// TwinCAT 3 PLC project IBF_System
// Title: IBF_System
// Company: Industrial Brains B.V.
// ProjectVersion: 0.0.0.0
// Description: system and module base functions
// ProgramVersion: 3.1.4023.0
// libraries:
//   IBF_Devices, * (Industrial Brains B.V.)
//   IBF_HMI, * (Industrial Brains B.V.)
//   IBF_Utilities, * (Industrial Brains B.V.)
//   Tc2_Standard, * (Beckhoff Automation GmbH)
//   Tc2_System, * (Beckhoff Automation GmbH)
//   Tc2_Utilities, * (Beckhoff Automation GmbH)
//   Tc3_Module, * (Beckhoff Automation GmbH)
// project tree:
//   GVLs/ PAR_System.TcGVL, GVL_System.TcGVL
//   / PlcTask.TcTTO
//   FaultHandler/ Fb_SystemFaultHandler.TcPOU (excluded from build)
//   ModuleBase/Base/ Fb_ModuleBase.TcPOU
//   SystemBase/DataTypes/ E_StateSystem.TcTLEO, Udt_ModuleId.TcDUT
//   SystemBase/ SystemBase.TcPOU
//   _TESTS/ FB_DummyModule.TcPOU, PRG_TEST.TcPOU

CONFIGURATION IBF_System
    RESOURCE PLC ON TwinCAT3
        TASK PlcTask(INTERVAL := T#10ms, PRIORITY := 6);
        PROGRAM PRG_TEST WITH PlcTask : PRG_TEST;
    END_RESOURCE
END_CONFIGURATION

// ---- SystemBase/DataTypes/E_StateSystem.TcTLEO
{attribute 'qualified_only'}
{attribute 'strict'}
{attribute 'to_string'}
TYPE E_StateSystem :
(
	FirstCycle		,
	CheckLogger		,
	CheckReferences ,  	// System is checking if module references are OK
	Initialize		, 	// System is initializing
	LoadParameters	, 	// System is loading parameters from/to file
	Safe			, 	// System is in safety state
	Enable			, 	// System is enabling 
	Home			, 	// system is homing 
	Resetting		, 	// System is resetting
	Idle			, 	// system is waiting for commands
	Manual			, 	// System is in manual mode
	SemiAuto		, 	// System is in semi auto mode
	Automatic		, 	// system is in automatic mode 
	Fault				// System is in Fault state
) UDINT;
END_TYPE

// ---- SystemBase/DataTypes/Udt_ModuleId.TcDUT
TYPE Udt_ModuleId :
STRUCT
	nNumber		: UDINT ; // Module identification number used for sorting order
	sName		: STRING; // Module name
	pFunction	: POINTER TO Fb_ModuleBase ;
END_STRUCT
END_TYPE

// ---- GVLs/PAR_System.TcGVL
{attribute 'qualified_only'}
VAR_GLOBAL CONSTANT
	LOG_FOLDER : STRING := ''; // Location for the log files
END_VAR

// ---- GVLs/GVL_System.TcGVL

{attribute 'qualified_only'} // Main system variables and state indicators
{attribute 'analysis':= '-33'}
VAR_GLOBAL CONSTANT
	cnMaxNUMBEROFMODULES 	: UDINT := 10 		; // "maximum" number of modules in the system
	CtAIRPRESSUREDELAY	: TIME 	:= T#500MS	; // Timout before air fault becomes active
	cbUPSPRESENT		: BOOL	:= FALSE 	; // Enable automatic shutdown when power is interupted
END_VAR
VAR_GLOBAL PERSISTENT
	nTotalUnitsProduced		: UDINT ; // Units produced 
END_VAR

// ---- _TESTS/PRG_TEST.TcPOU
PROGRAM INTERNAL PRG_TEST
VAR
 	bEnableTests : BOOL;

	fbDummyModule : FB_DummyModule;
END_VAR

IF bEnableTests THEN
	// SystemBase is the master program. it controls all underlying modules.
	SystemBase();

	// Call modules
	fbDummyModule(nModuleID:= 1);
END_IF

END_PROGRAM

// ---- _TESTS/FB_DummyModule.TcPOU
FUNCTION_BLOCK INTERNAL FB_DummyModule EXTENDS Fb_ModuleBase
VAR_INPUT
	// Inputs for testing module <> system interaction
	bAllowInit 		: BOOL;
	bAllowAutomatic : BOOL;
	bAllowSemiAuto 	: BOOL;
	bAllowHold 		: BOOL;
	bAllowHome 		: BOOL;
	bAllowReset 	: BOOL;
	bAllowIsSafe 	: BOOL;
	bAllowManual 	: BOOL;
END_VAR
VAR
	nCallsToExecAutomatic : ULINT;
	nCallsToExecHold : ULINT;
	nCallsToExecHome : ULINT;
	nCallsToExecInit : ULINT;
	nCallsToExecManual : ULINT;
	nCallsToExecReset : ULINT;
	nCallsToExecSafeStop : ULINT;
	nCallsToExecSemiAuto : ULINT;
END_VAR

SUPER^();

METHOD PROTECTED  CallComponents : BOOL
VAR_INPUT
END_VAR
END_METHOD

METHOD PROTECTED  CheckCollision : BOOL // Checks device commands for positble collisions  and block if necesarry
VAR_INPUT
END_VAR
END_METHOD

METHOD PROTECTED  ExecAutomatic : BOOL
VAR_INPUT
END_VAR
bAutomatic := bAllowAutomatic;
ExecAutomatic := bAutomatic;

nCallsToExecAutomatic := nCallsToExecAutomatic + 1;
END_METHOD

METHOD PROTECTED  ExecBaseFunctions : BOOL
VAR_INPUT
END_VAR
END_METHOD

METHOD PROTECTED  ExecEnable
VAR_INPUT
END_VAR
END_METHOD

METHOD PROTECTED  ExecHold : BOOL
VAR_INPUT
END_VAR
bHeld := bAllowHold;
ExecHold := bHeld;

nCallsToExecHold := nCallsToExecHold + 1;
END_METHOD

METHOD PROTECTED  ExecHome : BOOL
VAR_INPUT
END_VAR
bHomed := bAllowHome;
ExecHome := bHomed;

nCallsToExecHome := nCallsToExecHome + 1;
END_METHOD

METHOD PROTECTED  ExecIdle
VAR_INPUT
END_VAR
END_METHOD

METHOD PROTECTED  ExecInit : BOOL
VAR_INPUT
END_VAR
bInitialized := bAllowInit;
ExecInit := bInitialized;

nCallsToExecInit := nCallsToExecInit + 1;
END_METHOD

METHOD PROTECTED ExecManual : BOOL
VAR_INPUT
END_VAR
bManual := bAllowManual;

nCallsToExecManual := nCallsToExecManual + 1;
END_METHOD

METHOD PROTECTED  ExecReset : BOOL
VAR_INPUT
END_VAR
bResetDone := bAllowReset;
ExecReset := bResetDone;

nCallsToExecReset := nCallsToExecReset + 1;
END_METHOD

METHOD PROTECTED  ExecSafeStop : BOOL
VAR_INPUT
END_VAR
bIsSafe := bAllowIsSafe;
ExecSafeStop := bIsSafe;

nCallsToExecSafeStop := nCallsToExecSafeStop + 1;
END_METHOD

METHOD PROTECTED  ExecSemiAuto : BOOL
VAR_INPUT
END_VAR
bSemiAuto := bAllowSemiAuto;
ExecSemiAuto := bSemiAuto;

nCallsToExecSemiAuto := nCallsToExecSemiAuto + 1;
END_METHOD

END_FUNCTION_BLOCK

// ---- ModuleBase/Base/Fb_ModuleBase.TcPOU
{attribute 'reflection'}
FUNCTION_BLOCK PUBLIC ABSTRACT Fb_ModuleBase
VAR_INPUT
	nModuleID			: 	UINT 	:= 1 	; // module reference number used for fault, enable, reset, and safety functions (default := 1, 0 = main system)
	// main system Inputs
	bEnable				: 	BOOL	:= FALSE ; // (autolinked) module enable 	
	bCmdReset 			: 	BOOL	:= FALSE ; // (AutoLinked) reset all faults 
	bCmdPause			: 	BOOL 	:= FALSE ; // Pause command	bCmdToStart			
END_VAR
VAR_OUTPUT
	stIdentity			: UDT_Identity;
	bAddedToSystem		: BOOL 		:= FALSE 			; // module has been added to the system

	// Fault indications
	bReqPause		: BOOL := FALSE ; // Request for auto cycle pause
	bReqContinue	: BOOL := FALSE ; // Request for auto cycel continue
	// Check values
	bReferenceOk	: BOOL := FALSE ; // All module references  have been checked
	// State indication
	bIsSafe			: BOOL := FALSE ; // Module is safe and locked until safety is ok
	bInitialized	: BOOL := FALSE ; // Module startup initialized waiting for startup command
	bHomed 			: BOOL := FALSE ; // Module startup homed waiting for further further commands

	bHeld	 		: BOOL := FALSE ; // Module Hold Motion is held until command is released	
	
	bResetDone 		: BOOL := FALSE ; // Module reset is done   
	
	bManual 		: BOOL := FALSE ; // Module Work status Module in Manual
	bSemiAuto		: BOOL := FALSE ; // Module work status in semi automatic
	bStartAuto		: BOOL := FALSE ; // Module start automatic cycle 
	bAutomatic 		: BOOL := FALSE ; // Module Work status Module in Automatic mode
	bPaused			: BOOL := FALSE ; // Module paused
	bStopAuto		: BOOL := FALSE ; // Module Stop automatic
	bStopping		: BOOL := FALSE ; // MOdule stopping auto cycle
	
	bLocked			: BOOL := FALSE ; // module is locked for commands
END_VAR
VAR 
	// Internal functions 
	ReCmdReset 			: R_TRIG ;
	// Persistent data
	bCmdWritePersistent : BOOL := FALSE ; // write persistent data to memory
	// Module data
	stFault			: UDT_Fault			; // Message data
	// Function path 
	{attribute 'instance-path'} 
    {attribute 'noinit'}
	sPath				: STRING	; // Path name of function (used for manual reference)
END_VAR

// Get device name from function
IF stIdentity.sName = '' THEN 
	stIdentity.nId := nModuleID;
	stIdentity.sName := F_FBNameFromPath(sPath := sPath);
END_IF

// Add module to system
IF NOT bAddedToSystem THEN
	bAddedToSystem S= SystemBase.CmdAddModule(refToModule := THIS^);
	RETURN;
END_IF

IF NOT bReferenceOk THEN 
	bReferenceOk S= CheckReferences();
	RETURN;
ELSE 
	// Execute functions
	ExecMainBaseFunctions();
END_IF

// Reset pause request 
bReqPause 		R= bPaused ;
bReqContinue    R= NOT bPaused 	;

METHOD PROTECTED ABSTRACT CallComponents : BOOL
VAR_INPUT
END_VAR
END_METHOD

METHOD PROTECTED ABSTRACT CheckCollision : BOOL // Checks device commands for positble collisions  and block if necesarry
VAR_INPUT
END_VAR
END_METHOD

METHOD PUBLIC CheckReferences : BOOL
VAR_INPUT
END_VAR
bReferenceOk := TRUE;
END_METHOD

METHOD INTERNAL CmdAutomatic : BOOL
VAR_INPUT
END_VAR
// CmdAutomatic follows a different pattern than CmdSemiAuto, because Automatic mode can receive start/stop commands.
// Therefore, ExecAutomatic is called by ExecMainBaseFunctions instead of this method.
IF NOT bAutomatic THEN 
	bStartAuto 		:= TRUE ;
	bStopping		:= FALSE;
END_IF 

bSemiAuto	:= FALSE;
bManual		:= FALSE;

CmdAutomatic 	:= bAutomatic;
END_METHOD

METHOD INTERNAL CmdEnable
ExecEnable();

bSemiAuto	:= FALSE;
bAutomatic 	:= FALSE;
END_METHOD

METHOD INTERNAL CmdEstop : BOOL
VAR_INPUT
END_VAR
ExecSafeStop();
bSemiAuto	:= FALSE;
bAutomatic 	:= FALSE;
bManual		:= FALSE;

CmdEstop := bIsSafe ;
END_METHOD

METHOD INTERNAL CmdHold : BOOL
VAR_INPUT
END_VAR
ExecHold();

CmdHold := bHeld ;
END_METHOD

METHOD Internal CmdHome : BOOL
VAR_INPUT
END_VAR
ExecHome();

CmdHome := bHomed;
END_METHOD

METHOD INTERNAL CmdIdle
ExecIdle();

bSemiAuto	:= FALSE;
bAutomatic 	:= FALSE;
END_METHOD

METHOD INTERNAL CmdInit : BOOL
VAR_INPUT
END_VAR
ExecInit();

CmdInit := bInitialized;
END_METHOD

METHOD Internal CmdManual : BOOL
VAR_INPUT
END_VAR
ExecManual();

bSemiAuto	:= FALSE;
bAutomatic 	:= FALSE;

CmdManual := bManual;
END_METHOD

METHOD INTERNAL CmdSemiAuto : BOOL
VAR_INPUT
END_VAR
ExecSemiAuto();

bAutomatic 	:= FALSE;
bManual		:= FALSE;

CmdSemiAuto := bSemiAuto;
END_METHOD

METHOD INTERNAL CmdStopAutomatic : BOOL
VAR_INPUT
END_VAR
IF bAutomatic THEN 
	bStartAuto 		:= FALSE ;
	bStopAuto 		:= TRUE ;
END_IF 

CmdStopAutomatic 	:= NOT bAutomatic;
END_METHOD

METHOD PROTECTED ABSTRACT ExecAutomatic : BOOL
VAR_INPUT
END_VAR
END_METHOD

METHOD PROTECTED ABSTRACT ExecBaseFunctions : BOOL
VAR_INPUT
END_VAR
END_METHOD

METHOD PROTECTED ABSTRACT ExecEnable
VAR_INPUT
END_VAR
END_METHOD

METHOD ExecFaultHandling : BOOL
VAR_INPUT
END_VAR
// Call message function
	GVL_Utilities.fbFaultHandler.CmdAddFault( stFault := stFault, stIdentity);

// Call reset functions
	ReCmdReset( CLK := bCmdReset);
	
	IF ReCmdReset.Q THEN 
		bResetDone := FALSE ;
	ELSIF NOT bResetDone THEN 
		IF bInitialized THEN
			bResetDone := ExecReset() AND GVL_Utilities.fbFaultHandler.CmdReset();
		ELSE
			bResetDone := TRUE ;		
		END_IF
	END_IF
	
	bCmdReset := FALSE ;
END_METHOD

METHOD PROTECTED ABSTRACT ExecHold : BOOL
VAR_INPUT
END_VAR
END_METHOD

METHOD PROTECTED ABSTRACT ExecHome : BOOL
VAR_INPUT
END_VAR
END_METHOD

METHOD PROTECTED ABSTRACT ExecIdle
VAR_INPUT
END_VAR
END_METHOD

METHOD PROTECTED ABSTRACT ExecInit : BOOL
VAR_INPUT
END_VAR
END_METHOD

METHOD INTERNAL ExecMainBaseFunctions : BOOL
VAR_INPUT
END_VAR
// Call fault handling function 
ExecFaultHandling();

// Check for any Internal collisions
IF bInitialized THEN
	CheckCollision();
END_IF

// Call components 
CallComponents();

//// Run automatic function 
IF bStopAuto OR bStopping THEN 
	bStopping 	:= ExecAutomatic();
	bAutomatic  := FALSE;
	bStopAuto	:= FALSE;
	bStartAuto 	:= FALSE;
ELSIF bStartAuto OR bAutomatic THEN 
	bAutomatic 	:= ExecAutomatic();
	bStartAuto 	:= FALSE;
END_IF

// Run Base Functions 
IF bInitialized 
AND bEnable
AND bHomed 
AND NOT bManual THEN 
	ExecBaseFunctions();
END_IF

// Persistent data 
IF bCmdWritePersistent THEN 
	bCmdWritePersistent R= DataManager.FbPersistentManager.Write();
END_IF
END_METHOD

METHOD PROTECTED ABSTRACT ExecManual : BOOL
VAR_INPUT
END_VAR
END_METHOD

METHOD PROTECTED ABSTRACT ExecReset : BOOL
VAR_INPUT
END_VAR
END_METHOD

METHOD PROTECTED ABSTRACT ExecSafeStop : BOOL
VAR_INPUT
END_VAR
END_METHOD

METHOD PROTECTED ABSTRACT ExecSemiAuto : BOOL
VAR_INPUT
END_VAR
END_METHOD

END_FUNCTION_BLOCK

// ---- SystemBase/SystemBase.TcPOU
{attribute 'reflection'}
PROGRAM SystemBase // System base program, from here all modules are controlled and the system functions are called.
VAR_INPUT // System configuration settings
	bIcfAirCheckPresent	: BOOL := TRUE; // System is equipped with air pressure sensor 
END_VAR
VAR_OUTPUT
	// Check values
	bReferenceOk		: BOOL := FALSE ; // All module references  have been checked

	// State indication
	bIsSafe				: BOOL := FALSE ; // Module is safe and locked until safety is ok

	bInitializing		: BOOL := FALSE ; // Module startup initializing
	bInitialized		: BOOL := FALSE ; // Module startup initialized waiting for startup command
	
	bParametersLoaded 	: BOOL := FALSE ; // Parameters have been loaded from the file(s) 

	bIdle 				: BOOL := FALSE ; // Module startup Idle no commands active

	bEnabling 			: BOOL := FALSE ; // Module Startup enabeling 
	bEnabled 			: BOOL := FALSE ; // Module Startup Enabled
	
	bHoming				: BOOL := FALSE ; // Module startup homing back to base position and recalibrate
	bHomed 				: BOOL := FALSE ; // Module startup homed waiting for further further commands

	bHolding 			: BOOL := FALSE ; // Module Module Hold motion command executing
	bHeld	 			: BOOL := FALSE ; // Module Hold Motion is held until command is released	
	
	bResetting 			: BOOL := FALSE ; // Module Reset resetting error status
	bResetDone 			: BOOL := FALSE ; // Module reset is done   

	bManual 			: BOOL := FALSE ; // Module Work status Module in Manual 
	
	bStartSemiAuto		: BOOL := FALSE ; // Start semi automatic mode 
	bSemiAuto			: BOOL := FALSE ; // Module work status module in semi automatic
	
	bStartAuto			: BOOL := FALSE ; // Start automatic mode
	bAutomatic 			: BOOL := FALSE ; // Module Work status Module in Automatic mode
	bStopAuto			: BOOL := FALSE ; // Stop automatic mode
	bStoppingAuto		: BOOL := FALSE ; // Stopping automatic mode
	
	bCmdPause			: BOOL := FALSE ; // Pause all modules 
	bPaused 			: BOOL := FALSE ; // all modules are paused
	
	bModuleLocked		: BOOL := FALSE ; // a module is locked for commands
END_VAR
VAR
	// Logger & loghandlers
	fbLogHandler_TxtFile : FB_LogHandler_TxtFile(
								sLogFolder := PAR_System.LOG_FOLDER,
								sLogFilePrefix := 'Log_',
								sLogFileExtension := 'txt',
								nMaxLogFileSize := 256*1024, // 256kb is enough for at least 1000 lines. The HMI text editor should be able to handle this (tested on a TwinCAT/BSB VM).
								nMaxNumberOfLogFiles := 100 // 256kb * 100 = 25MB
							);
	fbLogHandler_RetainableList : FB_LogHandler_RetainableList;
	fbLogger : FB_Logger();
			
	// System inputs 
	ibPowerSupplyOk	 	AT%I*	: BOOL  ; // System Power supply is ok 
	fbAirpressureOk 			: Fb_DevDigitalInputFunctions  	; // system airpressure is ok

	// Air handling
	fbValveMainAirSupply		: FB_DevValve ; // Main air supply valve 
	toffMainAir					: TOF	:= (PT := T#500MS ); // Main air supply off delay
	bAirOk						: BOOL := FALSE ; // Air pressure is ok 
	
	// System HMI commands
	fbStartSemiAuto				: FB_DevHMIButton ; // HMI start semi automatic button 
	fbStartAuto					: FB_DevHMIButton ; // HMI start automatic button

	// System commands 
	fbCmdStartSystem		 	: FB_DevPushbuttonLight  		; // (re)start system input from button
	fbCmdStartAuto				: FB_DevPushbuttonLight			; // Start system automatic cycle
	fbCmdStopAuto				: FB_DevPushbuttonLight			; // Start system automatic cycle
	fbCmdReset		 			: FB_DevPushbuttonLight 		; // System reset
	
	// System state
	fbStateMachine				: FB_StateMachine;
	eStateSystem				: E_StateSystem := E_StateSystem.FirstCycle; // State of system
	
	// Set system variables
	fbSetSystemVariables		: Fb_SystemVariables ;
	
	// Local faults (always fatal)
	stFault						: UDT_Fault := (FaultType := E_FaultTypes.FF); 

 	// Module states
	nNumberOfModules			: UDINT := 0 ; // Number of modules added to the system 
	arpModules					: ARRAY [1..GVL_System.cnMaxNUMBEROFMODULES] OF Udt_ModuleId ; 

	// Power down system function
	fTrigPowerSupply			: F_TRIG ; // falling edge trigger for power supply
	ntShutDown					: NT_Shutdown ; // shutdown system function 
END_VAR
VAR // safety 
	// inputs 
	ibEstopOk 			AT%I*	: BOOL  ; // System emergency stop ok
	ibSafetyFBErr		AT%I*	: BOOL	; // The "FB Error" group signal
	ibSafetyComErr		AT%I*	: BOOL	; // The "Com Error" group signal
	
	// Outputs 
	qbSafetyErrAckn		AT%Q*	: BOOL ; // Safety error acknowledge
	qbRunSafety			AT%Q*	: BOOL ; // Run safety program
	qbResetSafety		AT%Q*	: BOOL ; // Reset safety program

	// safety Reset Timer	
	TofSafetyErrAck				: TOF := (PT := T#500MS); // Safety reset timer
END_VAR
VAR // Miscellaneous
	stIdentity 		: UDT_Identity := (sName := 'System');
	bCmdResetBusy 	: BOOL;
END_VAR

// Call system functions 
CallSystemFunctions();

// Execute fault handing
ExecFaultHandling();

// Handle UPS
ExecUPS();

// Execute safety control (controls E-Stop safety modules and enables air supply)
ExecSafetyControl();

// Call modules 
CallModules();

// Call manual control handler (must be done after calling modules, otherwise bCmdManual will toggle
IBF_Devices.GVL_Devices.fbManualController(bBlockManualMode := (eStateSystem <> E_StateSystem.Manual));

// Execute state machine
ExecSystemRun();

METHOD PRIVATE CallModules : BOOL
VAR
	i : UDINT ;
END_VAR
VAR
	AllAutomatic : BOOL ;
	Stopping : BOOL;
	bAllStopped : BOOL;
END_VAR
// set base conditions
bReferenceOk	:= TRUE ;
bIsSafe			:= TRUE ;
bIdle			:= TRUE ;	
bHeld			:= TRUE ;
bResetDone 		S= bResetting	;
bManual			:= TRUE	;
bSemiAuto		:= TRUE ;
bAutomatic		:= FALSE; // Reverse feedback 
AllAutomatic 	:= TRUE ;
bStoppingAuto	:= TRUE ;
bEnabled		S= bEnabling ;
bHomed 			:= TRUE;
bPaused 		:= TRUE;
bAllStopped     := TRUE;

// copy inputs to modules 
FOR i := 1 TO nNumberOfModules DO 
	// set system commands
	arpModules[i].pFunction^.bEnable			:= bEnabled			;
	arpModules[i].pFunction^.bCmdReset			:= bResetting		;
	arpModules[i].pFunction^.bCmdPause			:= bCmdPause		; 
	// Read state indications 
	bReferenceOk 	R= NOT arpModules[i].pFunction^.bReferenceOk; 
	bIsSafe 		R= NOT arpModules[i].pFunction^.bIsSafe;
	bEnabled 		R= NOT arpModules[i].pFunction^.bEnable;
	bHeld			R= NOT arpModules[i].pFunction^.bHeld;
	bResetDone		R= NOT arpModules[i].pFunction^.bResetDone;
	bManual			R= NOT arpModules[i].pFunction^.bManual;
	bSemiAuto		R= NOT arpModules[i].pFunction^.bSemiAuto;
	bHomed			R= NOT arpModules[i].pFunction^.bHomed;
	bPaused			R= NOT arpModules[i].pFunction^.bPaused;
	bModuleLocked	S= arpModules[i].pFunction^.bLocked			; // Module is locked for commands
	bCmdPause 		R= arpModules[i].pFunction^.bReqContinue	; // Request continue from module
	bCmdPause		S= arpModules[i].pFunction^.bReqPause		; // Request for pause from module
	bAutomatic		S= arpModules[i].pFunction^.bAutomatic 		; // Stay in automatic even when one module is in automatic
	AllAutomatic	R= NOT arpModules[i].pFunction^.bAutomatic	; // reset start automatic when al modules are in automatic operation
	bStoppingAuto	R= NOT arpModules[i].pFunction^.bStopping;

	Stopping		:= arpModules[i].pFunction^.bStopping;
	
	bAllStopped     := NOT Stopping AND NOT bAutomatic AND bAllStopped;
END_FOR

// Reset start inputs
	bEnabling		R= bEnabled 	;
	bHolding		R= bHeld 		;
	bResetting		R= bResetDone 	;
	bStartSemiAuto	R= bSemiAuto	;
	bHoming			R= bHomed 		;
	bStartAuto		R= AllAutomatic	; 
	bStopAuto		R= bAllStopped	;
	bCmdPause		R= NOT bAutomatic	;
END_METHOD

METHOD PRIVATE CallSystemFunctions : BOOL
// Update system variables 
fbSetSystemVariables();

// Run logger
fbLogger.Run();

// Call global parameter handler
GVL_Parameters.fbParameterHandler();

// Check air pressure
IF bIcfAirCheckPresent THEN
	fbAirpressureOk();
	bAirOk := fbAirpressureOk.bFcoDelay ;
ELSE
	bAirOk := TRUE ;
END_IF

// Execute button functions 
fbStartAuto		(tDelay	:= T#100MS, bEmbedded := TRUE);
fbStartSemiAuto (tDelay	:= T#100MS, bEmbedded := TRUE); 
fbCmdReset 		(tDelay	:= T#5000MS, bEmbedded := TRUE); 
fbCmdStartSystem(bEmbedded := TRUE);
fbCmdStartAuto	(bEmbedded := TRUE);
fbCmdStopAuto	(bEmbedded := TRUE);

// Reset button (lamp)
IF (GVL_Utilities.fbFaultHandler.nActiveFaults > 0) THEN
	IF GVL_Utilities.fbFaultHandler.arActiveFaultTypes[E_FaultTypes.FF] THEN
		// Fatal fault
		fbCmdReset.CmdOn() ;
	ELSIF GVL_Utilities.fbFaultHandler.arActiveFaultTypes[E_FaultTypes.CF] THEN
		// Cycle fault
		fbCmdReset.CmdBlinkSlow() ;
	ELSIF NOT GVL_Utilities.fbFaultHandler.arActiveFaultTypes[E_FaultTypes.OM] THEN
		// Warning
		fbCmdReset.CmdBlinkFast() ;
	END_IF
END_IF

// execute input functions
fbValveMainAirSupply(	bEnable			:= TRUE,
						refFbManualCtrl	:= IBF_Devices.GVL_Devices.fbManualController);
END_METHOD

METHOD PUBLIC CmdAddModule : BOOL
VAR_INPUT
	refToModule : REFERENCE TO Fb_ModuleBase ; // reference to module function
END_VAR
VAR
	bModuleAdded	: BOOL := FALSE;
	i 				: UDINT ; 
END_VAR
// Check if device is not already in the array 
FOR i:= 1 TO GVL_System.cnMaxNUMBEROFMODULES DO
	IF arpModules[i].pFunction = 0 THEN 
		nNumberOfModules:= i;
		EXIT;	
	ELSIF arpModules[i].sName = refToModule.stIdentity.sName THEN 
		bModuleAdded := TRUE ;
	END_IF 
END_FOR

// If device is not found add device to the list
IF NOT bModuleAdded AND nNumberOfModules >= 1 AND nNumberOfModules <= GVL_System.cnMaxNUMBEROFMODULES THEN
	arpModules[nNumberOfModules].nNumber 	:= refToModule.nModuleID;
	arpModules[nNumberOfModules].sName		:= refToModule.stIdentity.sName	;
	arpModules[nNumberOfModules].pFunction 	:= ADR(refToModule)		;	
	bModuleAdded := TRUE ;
END_IF

CmdAddModule := bModuleAdded ;
END_METHOD

METHOD CmdReset : BOOL
VAR_INPUT
END_VAR
eStateSystem := E_StateSystem.Resetting;

CmdReset := TRUE;
END_METHOD

METHOD PRIVATE ExecAutomatic : BOOL
VAR_INPUT
END_VAR
VAR
	i : UDINT ;
END_VAR
IF bStopAuto THEN 
	FOR i := 1 TO nNumberOfModules DO 
		arpModules[i].pFunction^.CmdStopAutomatic() ;
	END_FOR
ELSIF bStartAuto THEN 
	// Run automatic function in 
	FOR i := 1 TO nNumberOfModules DO 
		arpModules[i].pFunction^.CmdAutomatic() ;
	END_FOR
END_IF
	
ExecAutomatic := NOT bStartAuto;
END_METHOD

METHOD INTERNAL ExecEnable
VAR
	i : UDINT ;
END_VAR
bEnabling := TRUE;

// Run module enable function
FOR i := 1 TO nNumberOfModules DO 
	arpModules[i].pFunction^.CmdEnable() ;
END_FOR
END_METHOD

METHOD PRIVATE ExecFaultHandling
// Register system faults
GVL_Utilities.fbFaultHandler.CmdAddFault(stFault := stFault, stIdentity);

// Call global fault handler
GVL_Utilities.fbFaultHandler();

// Reset command
bCmdResetBusy S= fbCmdReset.bFeStatus;
IF bCmdResetBusy THEN
	bCmdResetBusy R= GVL_Utilities.fbFaultHandler.CmdReset();
END_IF
END_METHOD

METHOD PRIVATE ExecHoming : BOOL
VAR_INPUT
END_VAR
VAR
	i : UDINT ;
END_VAR
// Home all modules
FOR i := 1 TO nNumberOfModules DO 
	IF NOT arpModules[i].pFunction^.bHomed THEN 
		arpModules[i].pFunction^.CmdHome();
	END_IF
END_FOR
 
bHoming := NOT bHomed;
ExecHoming := bHomed;
END_METHOD

METHOD INTERNAL ExecIdle
VAR
	i : UDINT ;
END_VAR
fbCmdStartSystem.CmdBlinkSlow();

// Run module idle function
FOR i := 1 TO nNumberOfModules DO 
	arpModules[i].pFunction^.CmdIdle() ;
END_FOR
END_METHOD

METHOD PUBLIC ExecManual : BOOL
VAR
	i : UDINT ;
END_VAR
bEnabled := FALSE ;
FOR i := 1 TO nNumberOfModules DO 
	arpModules[i].pFunction^.CmdManual() ;
END_FOR

ExecManual := bManual;
END_METHOD

METHOD PRIVATE ExecSafeHold : BOOL
VAR_INPUT
END_VAR
VAR
	i : UDINT ;
END_VAR
// Hold all modules
bStartAuto		:= FALSE;

FOR i := 1 TO nNumberOfModules DO 
	arpModules[i].pFunction^.CmdHold();
END_FOR

ExecSafeHold := bHeld ;
END_METHOD

METHOD PRIVATE ExecSafeReset : BOOL
VAR_INPUT
END_VAR
END_METHOD

METHOD PRIVATE ExecSafeStop : BOOL
VAR_INPUT
END_VAR
VAR
	i : UDINT ;
END_VAR
bEnabling		:= FALSE;
bInitializing	:= FALSE;
bHoming			:= FALSE;
bStartAuto		:= FALSE;
bStartSemiAuto	:= FALSE;

// Module safe stop
IF bInitialized AND bReferenceOk THEN 
	FOR i := 1 TO nNumberOfModules DO 
		arpModules[i].pFunction^.CmdEstop();
	END_FOR
END_IF

// Shut down air supply once all modules are safe
IF bIsSafe THEN 
	fbValveMainAirSupply.CmdSafeStop();
END_IF
 
ExecSafeStop := bIsSafe ;
END_METHOD

METHOD PRIVATE ExecSafetyControl: BOOL
// Trigger system faults
// NOTES: some faults trigger a automatic safety circuit reset

// Not safe, until proven otherwise
stFault.Active := TRUE;
stFault.FaultType := E_FaultTypes.FF;

IF ibSafetyFBErr THEN 
	IF NOT qbRunSafety AND NOT TofSafetyErrAck.Q THEN 
		qbSafetyErrAckn := TRUE; 
	END_IF
	stFault.Description	:= 'Safety module function block error';

ELSIF ibSafetyComErr THEN
	IF NOT qbRunSafety AND NOT TofSafetyErrAck.Q THEN 
		qbSafetyErrAckn := TRUE ;
	END_IF
	stFault.Description	:= 'Safety module communication fault';

ELSIF (NOT ibEstopOk) AND (bInitialized OR bInitializing) THEN
	stFault.Description	:= 'Emergency stop pressed';

ELSIF (NOT bAirOk) AND (bInitialized OR bInitializing) THEN
	stFault.Description	:= 'Main air pressure low';
	
ELSE // Everything OK!
	stFault.Active := FALSE;
END_IF

// Show emergency overlay (a modal HMI overlay which blocks all HMI functionality)
// when a fault is active
IBF_HMI.GVL_HMI.fbHMIControl.sEmergencyText := stFault.Description;
IBF_HMI.GVL_HMI.fbHMIControl.bShowEmergencyOverlay	:= stFault.Active;

// Set safety system in run mode
IF NOT ibSafetyFBErr 
	AND NOT ibSafetyComErr
	AND bInitialized 
THEN 
	qbRunSafety := TRUE ;
ELSE 
	qbRunSafety := FALSE;
END_IF

// Reset safety faults
TofSafetyErrAck(IN := qbSafetyErrAckn);
qbSafetyErrAckn := FALSE ;
qbResetSafety := fbCmdReset.bFeStatus;

// Air pressure
toffMainAir(IN := ibEstopOk);
IF toffMainAir.Q THEN
	fbValveMainAirSupply.CmdOpen();
END_IF
END_METHOD

METHOD PUBLIC ExecSemiAuto : BOOL
VAR
	i : UDINT ;
END_VAR
// Run automatic function in 
FOR i := 1 TO nNumberOfModules DO 
	arpModules[i].pFunction^.CmdSemiAuto() ;
END_FOR

ExecSemiAuto := bSemiAuto;
END_METHOD

METHOD INTERNAL ExecSystemRun
VAR
	bError : BOOL; // An error is active (fatal fault or cycle fault)
	sDummyString : T_MaxString;
END_VAR
// Check if there are any high-prio faults
bError := GVL_Utilities.fbFaultHandler.arActiveFaultTypes[E_FaultTypes.CF] OR GVL_Utilities.fbFaultHandler.arActiveFaultTypes[E_FaultTypes.FF];

// Default home screen
IBF_HMI.GVL_HMI.fbHMIControl.eHomeScreen := E_BaseVisu.Idle;

// State machine
fbStateMachine(nState := eStateSystem);

// Log all system state changes
// NOTE: this is not required, but at least 1 log message must be added to initialize the logger
IF fbStateMachine.bStateChanged THEN
	fbLogger.DEBUG(CONCAT('System state changed to ', TO_STRING(eStateSystem)));
END_IF
 
CASE eStateSystem OF 
	E_StateSystem.FirstCycle:
		// Add log handlers
		sDummyString := PAR_System.LOG_FOLDER; // Suppress unused variable error (Beckhoff bug)
		fbLogger.AddLogHandler(fbLogHandler_TxtFile);
		fbLogger.AddLogHandler(fbLogHandler_RetainableList);
		eStateSystem 	:= E_StateSystem.CheckLogger;

	E_StateSystem.CheckLogger:
		// Check if log handlers have been initialized correctly
		IF fbLogHandler_TxtFile.bLoggerInitialized THEN
			eStateSystem 	:= E_StateSystem.CheckReferences;
		ELSIF fbLogHandler_TxtFile.bFault THEN
			stFault.Active := TRUE;
			stFault.FaultType := E_FaultTypes.OM;
			stFault.Description := CONCAT('Logger: ', fbLogHandler_TxtFile.sFaultDescription);
			eStateSystem 	:= E_StateSystem.CheckReferences;
		END_IF

	E_StateSystem.CheckReferences:
		IF bReferenceOk THEN
			eStateSystem := E_StateSystem.Initialize ;
		END_IF

	E_StateSystem.Initialize:
		IF Init() THEN
			eStateSystem := E_StateSystem.LoadParameters;
		END_IF

	E_StateSystem.LoadParameters:
		bParametersLoaded := GVL_Parameters.fbParameterHandler.Init();
		IF GVL_Parameters.fbParameterHandler.bFault THEN
			stFault.Active := TRUE;
			stFault.FaultType := E_FaultTypes.OW;
			stFault.Description := CONCAT('ParameterHandler: ', GVL_Parameters.fbParameterHandler.sFaultDescription);
			eStateSystem := E_StateSystem.Safe ;
		ELSIF bParametersLoaded THEN
			eStateSystem := E_StateSystem.Safe ;
		END_IF

	E_StateSystem.Safe:
		IF bIsSafe AND ibEstopOk THEN 
			IF bError THEN
				eStateSystem := E_StateSystem.Fault ;
			ELSE
				eStateSystem := E_StateSystem.Enable;
			END_IF
		ELSIF fbCmdReset.bFeStatus THEN
			eStateSystem	:= E_StateSystem.Resetting;
		ELSE 
			ExecSafeStop();
		END_IF

	E_StateSystem.Enable:
		ExecEnable();
		IF bError THEN
			eStateSystem := E_StateSystem.Fault;
		ELSIF GVL_HMI.fbHMIControl.bInScreenManual THEN
			eStateSystem := E_StateSystem.Manual ;
		ELSIF bEnabled THEN 
			fbCmdStartSystem.CmdBlinkFast();
			IF fbCmdReset.bFeStatus THEN
				eStateSystem := E_StateSystem.Resetting ;
			ELSIF fbCmdStartSystem.bFeStatus THEN
				eStateSystem := E_StateSystem.Home ;
			END_IF
		END_IF

	E_StateSystem.Home:	
		IF bError THEN
			eStateSystem := E_StateSystem.Fault;
		ELSIF fbCmdReset.bFeStatus THEN
			eStateSystem := E_StateSystem.Safe;			
		ELSIF ExecHoming() THEN
			eStateSystem := E_StateSystem.Idle;
		END_IF

	E_StateSystem.Resetting:
		IF NOT bResetDone THEN 
			bResetting S= TRUE ;
		ELSIF NOT bIsSafe THEN 
			eStateSystem := E_StateSystem.Safe ;
		ELSIF bError THEN
			IF NOT bCmdResetBusy THEN
				eStateSystem := E_StateSystem.Fault ;
			END_IF
		ELSIF bHomed AND bEnabled THEN
			eStateSystem := E_StateSystem.Idle ;
		ELSE 
			eStateSystem := E_StateSystem.Enable ;
		END_IF

	E_StateSystem.Idle:
		ExecIdle();
		IF bError THEN
			eStateSystem := E_StateSystem.Fault;
		ELSIF fbCmdReset.bFeStatus THEN
			eStateSystem := E_StateSystem.Resetting;			
		ELSIF GVL_HMI.fbHMIControl.bInScreenManual THEN 
			eStateSystem := E_StateSystem.Manual ;
		ELSIF fbCmdStartSystem.bFeStatus THEN 
			eStateSystem := E_StateSystem.SemiAuto ;
		END_IF

	E_StateSystem.Manual:
		IF bError THEN
			eStateSystem := E_StateSystem.Fault;
		ELSIF fbCmdReset.bFeStatus THEN
			eStateSystem := E_StateSystem.Safe;			
		ELSIF IBF_Devices.GVL_Devices.fbManualController.bActive THEN
			ExecManual();
		END_IF
		
		IF NOT GVL_HMI.fbHMIControl.bInScreenManual THEN
			EStateSystem := E_StateSystem.Enable;
		END_IF 

	E_StateSystem.SemiAuto:
		ExecSemiAuto();
		IBF_HMI.GVL_HMI.fbHMIControl.eHomeScreen := E_BaseVisu.SemiAutomatic;
		IF bError THEN
			eStateSystem := E_StateSystem.Fault;
		ELSIF fbCmdReset.bFeStatus THEN
			eStateSystem := E_StateSystem.Idle;			
		ELSIF (fbCmdStartAuto.bFeStatus 
			OR fbStartAuto.bFcoDelay 
			OR bAutomatic)
		AND NOT bModuleLocked THEN 
			bStartAuto 		:= TRUE ;
			bStopAuto 		:= FALSE;
			eStateSystem 	:= E_StateSystem.Automatic ;
		END_IF					

	E_StateSystem.Automatic:
		ExecAutomatic();
		IBF_HMI.GVL_HMI.fbHMIControl.eHomeScreen := E_BaseVisu.Automatic;
		IF bError THEN
			eStateSystem := E_StateSystem.Fault;
		ELSIF fbCmdReset.bFeStatus THEN
			eStateSystem := E_StateSystem.Safe;
		ELSIF bAutomatic THEN
			IF fbCmdStartSystem.bFeStatus THEN
				eStateSystem := E_StateSystem.Idle ;
			ELSIF fbCmdStopAuto.bFeStatus THEN
				bStopAuto := TRUE;
			ELSIF fbCmdStartAuto.bFeStatus OR GVL_Utilities.fbFaultHandler.arActiveFaultTypes[E_FaultTypes.MC] THEN  
				bCmdPause 	:= NOT bPaused ;
			END_IF
		ELSIF NOT bStartAuto AND NOT bStopAuto THEN 
			eStateSystem := E_StateSystem.SemiAuto ;
		END_IF
		
		// Start button light control
		IF bAutomatic THEN 
			fbCmdStartAuto.CmdOn();
		ELSE
			fbCmdStartAuto.CmdBlinkFast(); 				
		END_IF

	E_StateSystem.Fault:
		// Reset enable bits
		bEnabled := FALSE;
		bEnabling := FALSE;
	
		IF fbCmdReset.bFeStatus THEN
			bResetDone		:= FALSE ;
			eStateSystem 	:= E_StateSystem.Resetting ;
		ELSIF GVL_Utilities.fbFaultHandler.arActiveFaultTypes[E_FaultTypes.FF] THEN 
			ExecSafeStop();
		ELSIF GVL_Utilities.fbFaultHandler.arActiveFaultTypes[E_FaultTypes.CF] THEN 
			ExecSafeHold();	
		END_IF 
	ELSE 
		;		
END_CASE

bModuleLocked := FALSE ;

IBF_HMI.GVL_HMI.fbHMIControl.sStatusText := TO_STRING(eStateSystem);
END_METHOD

ACTION ExecUPS:
// If the system has an UPS, shutdown immediately if power goes down 
fTrigPowerSupply(CLK := ibPowerSupplyOk);
ntShutDown(START := GVL_System.cbUPSPRESENT AND fTrigPowerSupply.Q);
END_ACTION

METHOD PRIVATE Init : BOOL
VAR_INPUT
END_VAR
VAR
	i : UDINT ;
END_VAR
// initialize system functions
IF bIcfAirCheckPresent THEN
	fbAirpressureOk.Init	( 	nId 		:= 1,
								nParentId	:= 0 );
END_IF 

fbCmdReset.Init	(	nId 		:= 2,
							nParentId	:= 0 );

fbValveMainAirSupply.Init(	nId			:= 3,
							nParentId	:= 0,
							eResetState	:= E_ValveResetState.Res_Closed,
							eSafeState	:= E_ValveResetState.Res_Closed);

fbCmdStartSystem.Init	( 	nId 		:= 4,
							nParentId	:= 0 );

fbCmdStartAuto.Init		( 	nId 		:= 5,
							nParentId	:= 0 );

fbCmdStopAuto.Init		( 	nId 		:= 6,
							nParentId	:= 0 );
							
// Initialize all modules
bInitialized	:= TRUE ;
FOR i := 1 TO nNumberOfModules DO 
	IF NOT arpModules[i].pFunction^.bInitialized THEN 
		arpModules[i].pFunction^.CmdInit();
	END_IF
	bInitialized R= NOT arpModules[i].pFunction^.bInitialized;
 END_FOR
 
bInitializing 	:= NOT bInitialized ;
Init := bInitialized ;
END_METHOD

END_PROGRAM

// ---- FaultHandler/Fb_SystemFaultHandler.TcPOU
FUNCTION_BLOCK INTERNAL Fb_SystemFaultHandler
VAR_INPUT
	nNumberOfModules	: UDINT := 0; // Number of modules connected to the system fault handler
	bsystemInitialized	: BOOL 	; // System init is done
END_VAR
VAR_IN_OUT
	arpModules			: ARRAY [1..gvl_main.cnMaxNUMBEROFMODULES] OF Udt_ModuleId ;
END_VAR
VAR_OUTPUT
	// Fault types 
	bSystemFF			: BOOL 	:= FALSE	; // System fatal fault is active
	bSystemCF			: BOOL 	:= FALSE	; // System Cycle fault is active
	bSystemMC 			: BOOL 	:= FALSE	; // a missing condition is active 
	bSystemOM			: BOOL	:= FALSE	; // operator message is active
END_VAR
VAR
	// Message variables
	bCmdSnoozeMessage	: REFERENCE TO BOOL  	:= GVL_Message.bCmdSnoozeMessage; // Snooze message display
	arActiveFaults 		: REFERENCE TO ARRAY [0..Param_Messages.nMAX_MESSAGES_SHOWN] OF UDT_Fault := GVL_Message.arActiveFaults ; // Active faults overview for showing in HMI
	arOperatorMessages	: REFERENCE TO ARRAY [0..Param_Messages.nMAX_MESSAGES_SHOWN] OF STRING ; // Active operator messages
	arOldFaults 		: ARRAY [0..Param_Messages.nMAX_MESSAGES_SHOWN] OF UDT_Fault ; // Old faults overview for comparing to active
	arWriteToLog		: ARRAY [0..Param_Messages.nMAX_MESSAGES_SHOWN] OF UDT_Fault ; // Fault array for writing to log file 
	nNumberOfOM			: UDINT ; // number of active operator messages
	nShownOM			: UDINT ; // currently shown operator message
	// Message logging
	dToday				: DATE 	; 
	nWriteStep			: UDINT := 0 ;
	bWriteError			: BOOL 	; // write to file error occured
	nWriteErroId		: UDINT ; // write error id
	// Write variables
	sActFileName		: STRING;
	hFile				: UINT	:= 0;(* File handle of the source file *)
	sMessageString		: ARRAY [0..Param_Messages.nMESSAGE_COLUMNS] OF STRING (GVL_Parameters.MAX_CSV_FIELD_LENGTH); (* temporary parameter buffer to string*)
	sCSVLine			: T_MaxString := '';(* Single CSV text line (row, record), we are using string as record buffer (your are able to see created fields) *)
	sCSVField			: T_MaxString := '';(* Single CSV field value (column, record field) *)
END_VAR
VAR // functions 
	tofSnoozeMessages	: TOF ; // timer function for message snoozing
	tonOperatorMessageCycle : TON ; // Timer for cycling through operator messages
	// Log to file functions
	fbFileOpen		: FB_FileOpen	;(* Opens file *)
	fbFileClose		: FB_FileClose	;(* Closes file *)
	fbFileGets		: FB_FileGets	;(* Reads one record (line) *)
	fbFilePuts		: FB_FilePuts	;(* Writes one record (line) *)
	fbReader		: FB_CSVMemBufferReader;(* Helper function block used to parse CSV data bytes (single record line) *)
	fbWriter		: FB_CSVMemBufferWriter;(* Helper function block used to create CSV data bytes (single record line) *)
END_VAR 
VAR CONSTANT
	stEmptyMessageUdt : UDT_Fault := (	Active 			:= FALSE,
									FaultType 		:= E_FaultTypes.NA,
									MessageNumber	:= 0,
									LocationNumber	:= 0,
									Description 	:= '',
									LocationName	:= '',
									ComponentType	:= E_ComponentTypes.NA,
									StartTime		:= DT#2020-1-1-00:00:00,
									EndTime			:= DT#2020-1-1-00:00:00,
									FullFaultId		:= '0'	)  ;
END_VAR

IF nNumberOfModules > 0 THEN 
	// Check modules for active messages 
	CheckForModuleFaults();
END_IF

IF bsystemInitialized THEN
	// set system fault bits 
	ExecSetFaultBit(); 
	// Log faults when they are reset
	ExecMessageCompare();
	// Logfile writer 
	ExecWriteToLog();
END_IF

// Message Screen controller 
ExecScreenControl();

METHOD PRIVATE CheckForModuleFaults : BOOL // check all modules for faults and copy them to the main fault array
VAR
	// functional variables
	i 					: UDINT ;
	j 					: UDINT ;
	// temporary fault storage
	arTempFaults	: ARRAY [0..Param_Messages.nMAX_MESSAGES_SHOWN] OF UDT_Fault ; // internal fault array
	p				: UDINT	;
END_VAR
{warning disable C0371}
IF NOT __ISVALIDREF(arpModules) THEN
	RETURN;
END_IF

// reset number of operator messages
MEMSET(destAddr :=ADR(arOperatorMessages), fillByte := 0, n := SIZEOF(arOperatorMessages));
nNumberOfOM := 0;
// Go over modules to check for fault messages 
FOR i := 1 TO nNumberOfModules DO 
	// Check for active messages
	FOR j := 0 TO Param_Messages.nMAX_MESSAGES_SHOWN DO 
		IF arpModules[i].pFunction^.fbFaultHandler.arActiveFaults[j].FaultType = E_FaultTypes.OM THEN 
			arOperatorMessages[nNumberOfOM] := arpModules[i].pFunction^.fbFaultHandler.arActiveFaults[j].Description ;
			nNumberOfModules := MIN(nNumberOfOM + 1, Param_Messages.nMAX_MESSAGES_SHOWN);		
		ELSIF arpModules[i].pFunction^.fbFaultHandler.arActiveFaults[j].FaultType > E_FaultTypes.OM THEN 
			arTempFaults[p]:= arpModules[i].pFunction^.fbFaultHandler.arActiveFaults[j] ;
			p := MIN( p + 1, Param_Messages.nMAX_MESSAGES_SHOWN);
		ELSE
			EXIT ;
		END_IF
	END_FOR
END_FOR

arOldFaults		:= arActiveFaults 	;
arActiveFaults	:= arTempFaults 	;
{warning restore C0371}
END_METHOD

METHOD PRIVATE ExecMessageCompare : BOOL
VAR
	// functional variables
	i 			: UDINT ;
	j 			: UDINT ;
	bFaultFound : BOOL ;
	p			: UDINT;
END_VAR
// Check if any changes occured in the active faults
FOR i := 0 TO Param_Messages.nMAX_MESSAGES_SHOWN DO
	// break loop if fault is empty
	IF  arOldFaults[i].FaultType = E_FaultTypes.NA THEN  
		EXIT;
	ELSE
		// check if the fault is still active
		bFaultFound := FALSE; 
		FOR j := 0 TO Param_Messages.nMAX_MESSAGES_SHOWN DO
			IF arOldFaults[i].FullFaultId = arActiveFaults[j].FullFaultId THEN
				bFaultFound := TRUE;
				EXIT;
			END_IF
		END_FOR
		// if the fault is not faund then wrtie it to the logging array for loging
		IF NOT bFaultFound THEN 
			arWriteToLog[p] := arOldFaults[i] ;
			p := p + 1 ; 
		END_IF
	END_IF
END_FOR

ExecSortMessages();
END_METHOD

METHOD PRIVATE ExecScreenControl : BOOL // Control message screen 
VAR_INPUT
END_VAR
tofSnoozeMessages(IN := bCmdSnoozeMessage, PT := GVL_Message.tMESSAGESNOOZEDURATION);

// Set screen control 
IF bSystemCF OR bSystemFF THEN 
	GVL_Message.bHideFaults := FALSE ;
	GVL_Message.bHideReset	:= FALSE ; 
ELSIF bSystemMC AND NOT tofSnoozeMessages.Q THEN 
	GVL_Message.bHideFaults := FALSE ;
ELSE
	GVL_Message.bHideFaults := TRUE ;
	GVL_Message.bHideReset	:= TRUE ; 
END_IF

// Cycle through operator messages
tonOperatorMessageCycle(PT := Param_Messages.tOMCYCLETIME, IN := NOT tonOperatorMessageCycle.Q);
IF tonOperatorMessageCycle.Q THEN
	IF nNumberOfOM > 0 THEN
		nShownOM := (nShownOM + 1) MOD nNumberOfOM;
		GVL_Message.sOPeratorMessage := arOperatorMessages[nShownOM];
	ELSE
		GVL_Message.sOPeratorMessage := '';
	END_IF
END_IF
END_METHOD

METHOD PRIVATE ExecSetFaultBit : BOOL
VAR
	// functional variables
	i 			: UDINT ;
END_VAR
bSystemFF	:= FALSE ;
bSystemCF	:= FALSE ;
bSystemMC	:= FALSE ;

FOR i := 0 TO Param_Messages.nMAX_MESSAGES_SHOWN DO
	bSystemFF	:= arActiveFaults[i].FaultType = E_FaultTypes.FF OR bSystemFF;
	bSystemCF	:= arActiveFaults[i].FaultType = E_FaultTypes.CF OR bSystemCF;
	bSystemMC	:= arActiveFaults[i].FaultType = E_FaultTypes.MC OR bSystemMC;
	bSystemOM	:= arActiveFaults[i].FaultType = E_FaultTypes.OM OR bSystemOM;
END_FOR
END_METHOD

METHOD INTERNAL ExecSortMessages : BOOL
VAR
	i : UDINT ;
	k : UDINT ;
	stTempMessageStorage : UDT_Fault ; // Temporary message storage for sorting
END_VAR
FOR k := 1 TO Param_Messages.nMAX_MESSAGES_SHOWN - 1 DO 
	FOR i := 0 TO Param_Messages.nMAX_MESSAGES_SHOWN - 2 DO 
		IF arActiveFaults[i].FaultType < arActiveFaults[i+1].FaultType THEN 
			stTempMessageStorage 	:= arActiveFaults[i];
			arActiveFaults[i]		:= arActiveFaults[i+1];
			arActiveFaults[i+1]		:= stTempMessageStorage;
		END_IF
	END_FOR	 
END_FOR

ExecSortMessages := TRUE;
END_METHOD

METHOD PRIVATE ExecWriteToLog : BOOL
VAR 
	i : UDINT ; 
	p : UDINT ; // Fault array pointer
END_VAR
dToday := DT_TO_DATE(Sys_Variables.SystemTime);
// create file name with Current date 
sActFileName 	:= CONCAT(STR1 := Param_Messages.sLOGFILE_PATH	, STR2 := Param_Messages.sLOGFILE_NAME	);
sActFileName 	:= CONCAT(STR1 := sActFileName					, STR2 := DATE_TO_STRING(dToday)		);
sActFileName 	:= CONCAT(STR1 := sActFileName					, STR2 := '.csv'						);

// ===== Start file write =====
CASE nWriteStep OF
	0:	(* Wait until log array is filled *)
		IF arWriteToLog[0].FaultType <> E_FaultTypes.NA THEN 
			hFile				:= 0;
			nWriteStep 			:= 1;
		ELSE 
			RETURN ;
		END_IF
	1:	(* Open source file *)
		fbFileOpen(  bExecute := FALSE  );
		fbFileOpen( sNetId := GVL_Parameters.sNetId, sPathName := sActFileName , nMode := FOPEN_MODEAPPEND OR FOPEN_MODETEXT,(* Open file in TEXT mode! *)
					ePath := PATH_GENERIC, bExecute := TRUE );
		nWriteStep := nWriteStep + 1 ;
	2:(* Wait until open not busy *)
		fbFileOpen( bExecute := FALSE, bError => bWriteError, nErrID => nWriteErroId, hFile => hFile );
		IF NOT fbFileOpen.bBusy THEN
			IF NOT fbFileOpen.bError THEN
				nWriteStep := nWriteStep + 1 ;
			ELSE(* Error: file not found? *)
				nWriteStep := 100;
			END_IF
		END_IF
	3: (* Check if faultrecord is active if so skip record *)
		nWriteStep := nWriteStep + 1 ;
	4:(* Convert one PLC record to CSV format *)
		sCSVLine := '';
		fbWriter.eCmd := eEnumCmd_First;(* Write first field value *)
		// write message data to string
		sMessageString[0] 	:= TO_STRING(arWriteToLog[p].FaultType				);
		sMessageString[1]	:= DT_TO_STRING(arWriteToLog[p].StartTime			);
		sMessageString[2]	:= DT_TO_STRING(Sys_Variables.SystemTime			);
		sMessageString[3]	:= UDINT_TO_STRING(arWriteToLog[p].MessageNumber	);
		sMessageString[4]	:= UDINT_TO_STRING(arWriteToLog[p].LocationNumber	); 
		sMessageString[5]	:= arWriteToLog[p].Description						;
		sMessageString[6]	:= arWriteToLog[p].LocationName						;
		sMessageString[7]	:= TO_STRING(arWriteToLog[p].ComponentType			);
		// write data to .csv buffer 
		FOR i := 0 TO Param_Messages.nMESSAGE_COLUMNS BY 1 DO
			sCSVField := STRING_TO_CSVFIELD(in :=  sMessageString[i], FALSE );
			(* Add new field to the record buffer *)
			fbWriter( 	pBuffer := ADR( sCSVLine ), cbBuffer := SIZEOF( sCSVLine ) - 1, putValue := sCSVField, pValue := 0, cbValue := 0,
						bCRLF := ( i = Param_Messages.nMESSAGE_COLUMNS ) );(* bCRLF == TRUE => Write CRLF after the last field value *)
			IF fbWriter.bOk THEN
				fbWriter.eCmd := eEnumCmd_Next;
			ELSE
				nWriteStep := 100;
				RETURN;
			END_IF
		END_FOR(* FOR nColumn := 0... *)

		(* FB_FilePuts adds allready CR (carriage return) to the written line.
		We have to replace the $R$L characters with $L character to avoid double CR. *)
		IF RIGHT( sCSVLine, 2 ) = '$R$L' THEN
			sCSVLine := REPLACE( sCSVLine, '$L', 2, LEN( sCSVLine ) - 1 );
		END_IF
		nWriteStep := nWriteStep + 1 ;
	5:	(* Write single text line to file *)
		fbFilePuts( bExecute := FALSE );
		fbFilePuts( sNetId := GVL_Parameters.sNetId, hFile := hFile, sLine := sCSVLine, bExecute := TRUE );
		nWriteStep := nWriteStep + 1 ;
	6:(* Wait until write not busy *)
		fbFilePuts( bExecute := FALSE, bError => bWriteError, nErrID => nWriteErroId );
		IF NOT fbFilePuts.bBusy THEN
			IF NOT fbFilePuts.bError THEN
				nWriteStep := nWriteStep + 1 ;
			ELSE(* Error *)
				nWriteStep := 100;
			END_IF
		END_IF
	7: (* clear fault from array and go to next fault *)
		arWriteToLog[p]:= stEmptyMessageUdt;
		IF p < Param_Messages.nMAX_MESSAGES_SHOWN THEN 
			p := p +1 ;
		END_IF
		nWriteStep := nWriteStep +1 ;
	8: (* If fault is active then repeat previous step, else close file*)		
		IF  arWriteToLog[p].FaultType <> E_FaultTypes.NA THEN 
			nWriteStep := 3 ;
		ELSE
			nWriteStep := 10;
		END_IF
	10:	(* Close source file *)
		fbFileClose( bExecute := FALSE );
		fbFileClose( sNetId := GVL_Parameters.sNetId, hFile := hFile, bExecute := TRUE );
		nWriteStep := 11;
	11:(* Wait until close not busy *)
		fbFileClose( bExecute := FALSE, bError => bWriteError, nErrID => nWriteErroId );
		IF ( NOT fbFileClose.bBusy ) THEN
			hFile 		:= 0;
			nWriteStep 	:= 100;
		END_IF
	100: (* Error or ready nWriteStep => cleanup *)
		IF ( hFile <> 0 ) THEN
			nWriteStep	:= 10; (* Close the source file *)
		ELSE
			nWriteStep 	:= 0;	(* Ready *)
			ExecWriteToLog := TRUE ;
		END_IF
END_CASE
END_METHOD

END_FUNCTION_BLOCK
